Fanuc KAREL source: ko00076.KL

-- PROVISIONAL review KL for V1013-1; original PC SHA256 f812351c044484a7ef9822a75f6f34424ff52e164639aacf0b6f8a7961637f54
-- Incomplete behavior may be omitted. Consult companion uncertainty JSON. Do not deploy.
PROGRAM KO00076
%NOLOCKGROUP
BEGIN
  -- UNRESOLVED_PC offsets 5-12; opcodes 9D,23
  -- UNRESOLVED_PC offsets 17-66; opcodes 27,22,1C,27,49,7E,AD,22,31,7E,4A
  -- UNRESOLVED_PC offsets 71-75; opcodes 7F
END KO00076
